FUNCTION_BLOCK OF_E_TimeOut (* Simple implementation of the timeout services *)
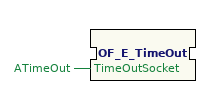
  SOCKETS
    TimeOutSocket : iec61499::events::ATimeOut;
  END_SOCKETS
END_FUNCTION_BLOCK
